{attribute 'GeneratedUsingTerminal: ER6001-0002-0016'}
{attribute addProperty BoxType "ER6001-0002-0016"}
{attribute addProperty Id "CtrlAT %Q*UINT2Data_OutAT %Q*ARRAY[0..21] OF USINT22"}
{attribute addProperty CRC "875731620"}
{attribute addProperty Size "24"}
TYPE COM_Outputs_5D00B5E7 :
STRUCT
	{attribute addProperty Name "Ctrl"}
	Ctrl AT %Q* : UINT;
	{attribute addProperty Name "Data_Out"}
	Data_Out AT %Q* : ARRAY[0..21] OF USINT;
END_STRUCT
END_TYPE

(* stored: Version 1.2.0.0, ProductVersion 3.1.4024.9
   DUT COM_Outputs_5D00B5E7: Id {7d3c7185-27a5-48fa-96f2-18da36835a57} *)
